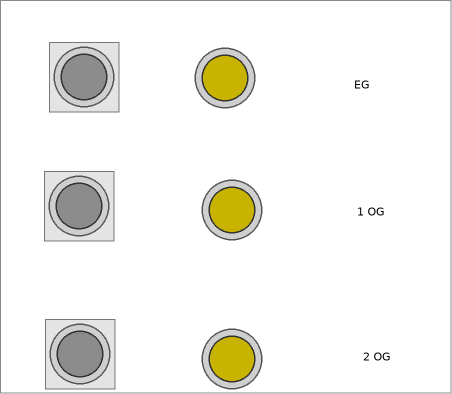
VISUALIZATION Visualization  // 452x394
    PushSwitch (49,42 70x70), variable: GVL.BP_EG, behaviour: TOGGLE, style: Switch-PushSwitch-Gray
    PushSwitch (44,171 70x70), variable: GVL.BP_1OG, behaviour: TOGGLE, style: Switch-PushSwitch-Gray
    PushSwitch (45,319 70x70), variable: GVL.BP_2OG, behaviour: TOGGLE, style: Switch-PushSwitch-Gray
    Label (287,70 150x30), "EG"
    Label (296,197 150x30), "1 OG"
    Label (302,342 150x30), "2 OG"
    Lamp1 (190,43 70x70), variable: GVL.Lampe_EG, style: Lamp-Lamp1-Yellow
    Lamp1 (197,175 70x70), variable: GVL.Lampe_1OG, style: Lamp-Lamp1-Yellow
    Lamp1 (197,324 70x70), variable: GVL.Lampe_2OG, style: Lamp-Lamp1-Yellow
END_VISUALIZATION

(* stored: Version 1.1.0.1, ProductVersion 3.1.4024.16
   Visu Visualization: Id {1e4210f6-ae84-47c1-b7ad-2a404f4ed338} *)
